# EPICS substitutions: gigeApp/Db/pluginMJPG.substitutions
#
# pluginMJPG.substitutions
#

file NDPluginBase.template
{
	{
	P=$(CAM):,
	R=MJPG$(N):,
	PORT=MJPG$(N),
	ADDR=0,
	TIMEOUT=1,
	NDARRAY_PORT=$(PLUGIN_SRC),
	NDARRAY_ADDR=0
	}
}

# Macros:
#  P        Device Prefix
#  R        Device Suffix
#  PORT     Asyn Port name
#  QUALITY  Jpeg Quality in percent
#  MAXW     Maximum Jpeg Width
#  MAXH     Maximum Jpeg Height
file ffmpegStream.template
{
	{
	P=$(CAM):,
	R=MJPG$(N):,
	PORT=MJPG$(N),
	QUALITY=100,
	}
}
